FUNCTION_BLOCK FB_BWK_SchreibeDaten
VAR_INPUT
	WP_Stellung : BOOL;
END_VAR
VAR_OUTPUT
	OUT_WP_Stellung : BOOL;
END_VAR
VAR
END_VAR

OUT_WP_Stellung := WP_Stellung;

END_FUNCTION_BLOCK

(* stored: Version 1.1.0.1, ProductVersion 3.1.4024.9
   POU FB_BWK_SchreibeDaten: Id {dcd11783-e60e-452e-b231-84e49a9b4f16}, SpecialFunc None *)
